//----------------------------------------------------------------------------//
//            Copyright 2018 Rieckermann Engineering Operations               //
//----------------------------------------------------------------------------//
// Description:                                                               //
// This file contains globally addressable event flags and data. The function //
// traverses the event datablock UDT structures to see if any event bits have //
// been raised. This is called each scan from the main program block OB1      //
// which therefore takes care of the looping required.                        //
//----------------------------------------------------------------------------//
// Revision history:                                                          //
// Rev By               Date        CC        Note                            //
// 1.0 David Paspa      29-Jun-2018 NA        Reboot design for S7-1500 from  //
//                                            ifbEventPrompt.                 //
//----------------------------------------------------------------------------//
FUNCTION_BLOCK "ifbEventLogMsg"
TITLE = S7 Alarms for SFC log messages
{ S7_Optimized_Access := 'TRUE' }
AUTHOR : REO
NAME : ifbEventLogMsg
VERSION : 1.0

//----------------------------------------------------------------------------//
// Declare variables:                                                         //
//----------------------------------------------------------------------------//
@@TEMPLATE_BEGIN@@
VAR
@@ATTR_BEGIN|pEventLogMsgNum@@
    eventLogMsg : Array[1..@@IDXEVENTMAX@@] of "udtEventLogMsg";   // SFC events for logging messages
@@ATTR_END|pEventLogMsgNum@@
@@ATTR_BEGIN|pEventLogMsgAll@@
    Program_Alarm_@@IDXEVENT@@ : Program_Alarm;
@@ATTR_END|pEventLogMsgAll@@
@@ATTR_BEGIN|pEventLogMsgAll@@
    Alarm@@IDXEVENT@@_ErrorBit1 : Bool;
    Alarm@@IDXEVENT@@_ErrorBit2 : Bool;
    Alarm@@IDXEVENT@@_StatusWord1 : Word;
    Alarm@@IDXEVENT@@_StatusWord2 : Word;
    Alarm@@IDXEVENT@@_StateByte : Byte;
@@ATTR_END|pEventLogMsgAll@@
	SourceData : Word;
END_VAR

VAR_TEMP
    almError : Bool;
    almState : Byte;
    almStatus : Word;
END_VAR

BEGIN
@@ATTR_BEGIN|pEventLogMsgAll@@
NETWORK
TITLE = Raise message event if required
    //------------------------------------------------------------------------//
    // EVENT   EVENT   EVENT   EVENT   EVENT   EVENT   EVENT   EVENT   EVENT  //
    // EVENT   EVENT   EVENT   EVENT   EVENT   EVENT   EVENT   EVENT   EVENT  //
    //                                                                        //
    // Raise the simple message event if requested. No acknowledge required:  //
    //------------------------------------------------------------------------//
    L @@IDXEVENT@@;
    T #SourceData;

    CALL #Program_Alarm_@@IDXEVENT@@
    (   SIG       := #eventLogMsg[@@IDXEVENT@@].trigger ,
		SD_1      := #SourceData ,
        Error     := #Alarm@@IDXEVENT@@_ErrorBit1 ,
        Status    := #Alarm@@IDXEVENT@@_StatusWord1
    );

@@ATTR_END|pEventLogMsgAll@@

@@TEMPLATE_END@@
END_FUNCTION_BLOCK
